// TIA Portal V17 export
// export: Created 2022-07-20T06:59:44.8939204Z, ExportSetting WithDefaults, DisplayName Totally Integrated Automation Portal, DisplayVersion V17, DisplayName TIA Portal Openness, DisplayVersion V17, DisplayName TIA Portal Version Control Interface, DisplayVersion V17, DisplayName SINAMICS Startdrive Advanced, DisplayVersion V17, DisplayName SINAMICS Startdrive G130, G150, S120, S150, SINAMICS MV, S210, DisplayVersion V17, DisplayName SINAMICS Startdrive G110M, G120, G120C, G120D, G120P, G115D, DisplayVersion V17, DisplayName STEP 7 Professional, DisplayVersion V17, DisplayName STEP 7 Safety, DisplayVersion V17, DisplayName WinCC Advanced, DisplayVersion V17
FUNCTION "FC10072_ScalingAirExtraction_VolatgeFeedback" : Void   // FC10072, LAD
{ S7_Optimized_Access := 'TRUE' }
VERSION : 0.1
// stored: AutoNumber false, IsIECCheckEnabled false, SetENOAutomatically false, UDAEnableTagReadback false
   VAR_INPUT
      VoltageFeedback : Real;
      X_UVPower_Min : Real;   // 0-100%
      X_UVPower_Max : Real;   // 0-100%
      Y_AirPower_Min : Real;   // 0-100%
      Y_AirPower_Max : Real;   // 0-100%
      PWM_Minimum : Real;
      PWM_Maximum : Real;   // Frequence
   END_VAR
   VAR_OUTPUT
      Analogical_Value : Int;
      PWM_FrequenceValue : Real;
   END_VAR
   VAR_TEMP
      Analogical_ValueTemp : Real;
   END_VAR
BEGIN

REGION Network 1 (SCL): Generate the PWM Air Extractor SetPoint
   IF #VoltageFeedback < #X_UVPower_Min THEN
       #PWM_FrequenceValue := 0;
       #Analogical_Value := 0;
   ELSIF #VoltageFeedback > #X_UVPower_Max THEN
       #PWM_FrequenceValue := #Y_AirPower_Max * #PWM_Maximum / 100;
       #Analogical_Value := REAL_TO_INT(#Y_AirPower_Max * 27648 / 100);
   ELSE
       "FC10020_Linearization"(X1 := #X_UVPower_Min,
                               Y1 := #Y_AirPower_Min * #PWM_Maximum / 100,
                               X2 := #X_UVPower_Max,
                               Y2 := #Y_AirPower_Max * #PWM_Maximum / 100,
                               X := #VoltageFeedback,
                               Y => #PWM_FrequenceValue);
       "FC10020_Linearization"(X1 := #X_UVPower_Min,
                               Y1 := #Y_AirPower_Min * 27648 / 100,
                               X2 := #X_UVPower_Max,
                               Y2 := #Y_AirPower_Max * 27648 / 100,
                               X := #VoltageFeedback,
                               Y => #Analogical_ValueTemp);
       #Analogical_Value := REAL_TO_INT(#Analogical_ValueTemp);
   END_IF;
END_REGION
END_FUNCTION
